FUNCTION_BLOCK RejectWithMessageAsyncHandler IMPLEMENTS I_AsynchronousRpcHandler
VAR
END_VAR

METHOD Handle
VAR_INPUT
	Parameters : I_Deserializer;
	Response : I_AsynchronousRpcResponse;
END_VAR
VAR
END_VAR
Response.RejectWithError('EXAMPLE_ERROR_CODE','This is the reject message');
END_METHOD

END_FUNCTION_BLOCK

(* stored: Version 1.1.0.1, ProductVersion 3.1.4024.15
   POU RejectWithMessageAsyncHandler: Id {76f722c4-335d-4072-b575-36ba2411bf2a}, SpecialFunc None
   Method Handle: Id {6cced2f9-9720-439e-8ec3-902320a03d64} *)
